(* PLC project pro1003, at09 pro1003 1 *)
(* stored: creationDateTime 2023-04-16T15:18:15, productRelease 0, modificationDateTime 2023-05-21T16:46:51, version 1, language ru-RU *)

(* LED Control *)
PROGRAM prog_led
  VAR_EXTERNAL
    LED_USER : BOOL;
    STATE_REGUL : WORD;
  END_VAR
  VAR
    TONb0 : TONb;
  END_VAR

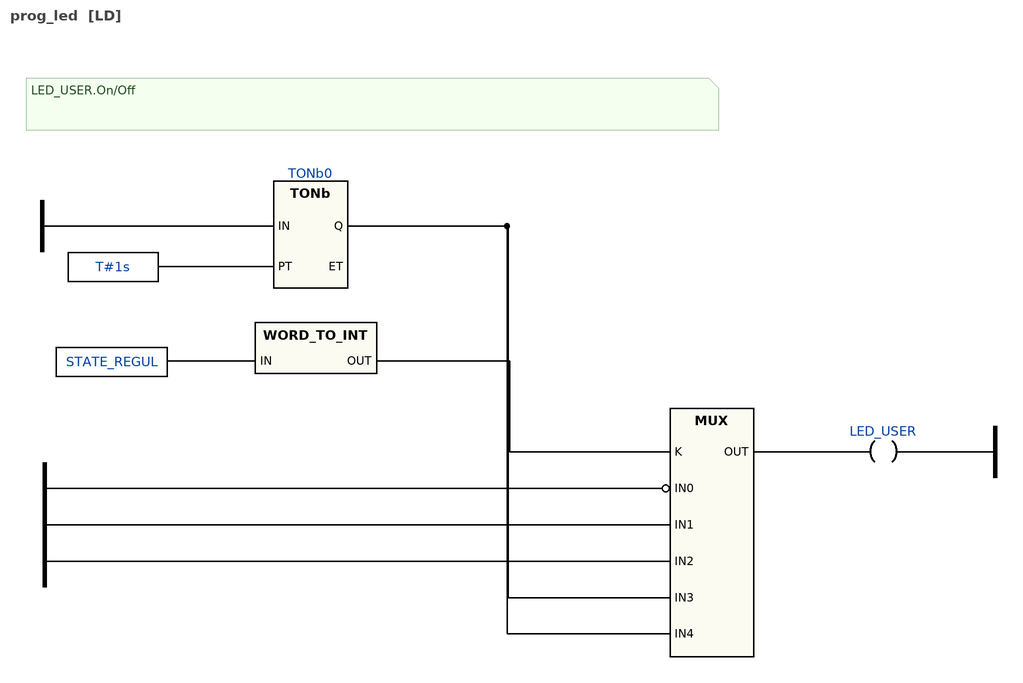
(* LD diagram, written out as Structured Text *)
(* LED_USER.On/Off *)
TONb0(IN := TRUE, PT := T#1s);
LED_USER := MUX(WORD_TO_INT(STATE_REGUL), NOT TRUE, TRUE, TRUE, TONb0.Q, TONb0.Q);
END_PROGRAM

(* Button Control *)
PROGRAM prog_button
  VAR_EXTERNAL CONSTANT
    HS_001_DIn : BYTE;
    HS_002_DIn : BYTE;
  END_VAR
  VAR CONSTANT
    DIMode_Norm : BYTE := 1;  (* DI.Mode (Normal) *)
  END_VAR
  VAR
    DIMode0 : DIMode;
    DIMode1 : DIMode;
  END_VAR

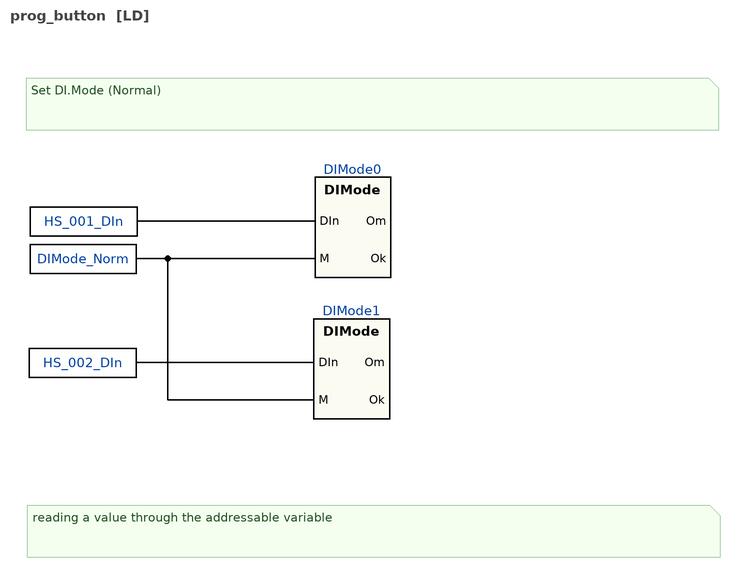
(* LD diagram, written out as Structured Text *)
(* Set DI.Mode (Normal) *)
DIMode0(DIn := HS_001_DIn, M := DIMode_Norm);
DIMode1(DIn := HS_002_DIn, M := DIMode_Norm);
(* reading a value through the addressable variable *)
END_PROGRAM

(* Sensor Control *)
PROGRAM prog_sensor
  VAR_EXTERNAL CONSTANT
    TT_001_AIn : BYTE;
    TT_MCU_AIn2 : BYTE;
  END_VAR
  VAR CONSTANT
    AIMode_Tmp36 : BYTE := 11;  (* AI.Mode (TMP36) *)
    AIMode_TmpMcu : BYTE := 12;  (* AI.Mode (TMP_MCU) *)
  END_VAR
  VAR
    AIMode0 : AIMode;
    AIMode1 : AIMode;
  END_VAR

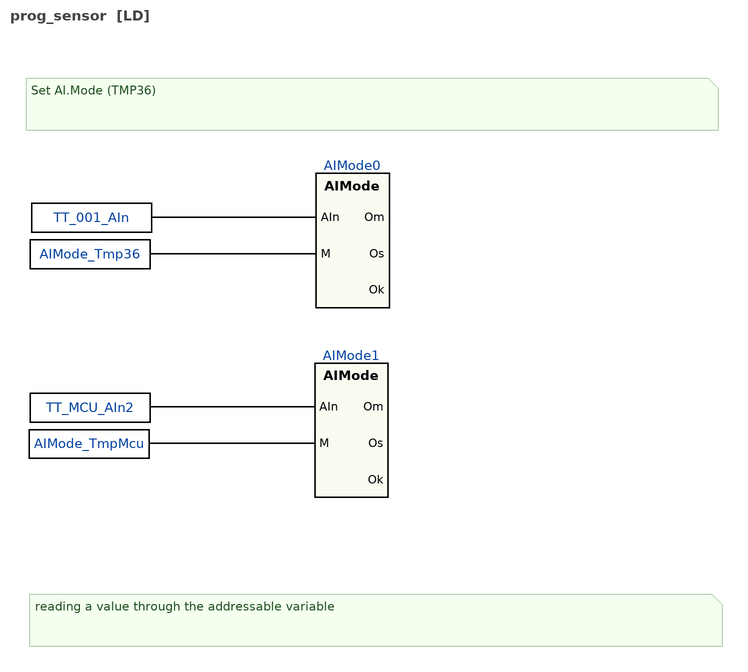
(* LD diagram, written out as Structured Text *)
(* Set AI.Mode (TMP36) *)
AIMode0(AIn := TT_001_AIn, M := AIMode_Tmp36);
AIMode1(AIn := TT_MCU_AIn2, M := AIMode_TmpMcu);
(* reading a value through the addressable variable *)
END_PROGRAM

(* Output Control *)
PROGRAM prog_output
  VAR_EXTERNAL CONSTANT
    H_001_DOn : BYTE;
  END_VAR
  VAR_EXTERNAL
    H_001_V : BOOL;
  END_VAR
  VAR_EXTERNAL CONSTANT
    C_001_DOn : BYTE;
  END_VAR
  VAR_EXTERNAL
    C_001_V : BOOL;
    STATE_REGUL : WORD;
    HEAT : BOOL;
  END_VAR
  VAR CONSTANT
    DOMode_Norm : BYTE := 1;  (* DO.Mode (Normal) *)
  END_VAR
  VAR
    DOMode0 : DOMode;
    DOMode1 : DOMode;
  END_VAR
  VAR  (* added by the conversion: wires and edge detectors of the diagram *)
    _WORD_TO_INT26_OUT : INT;
  END_VAR

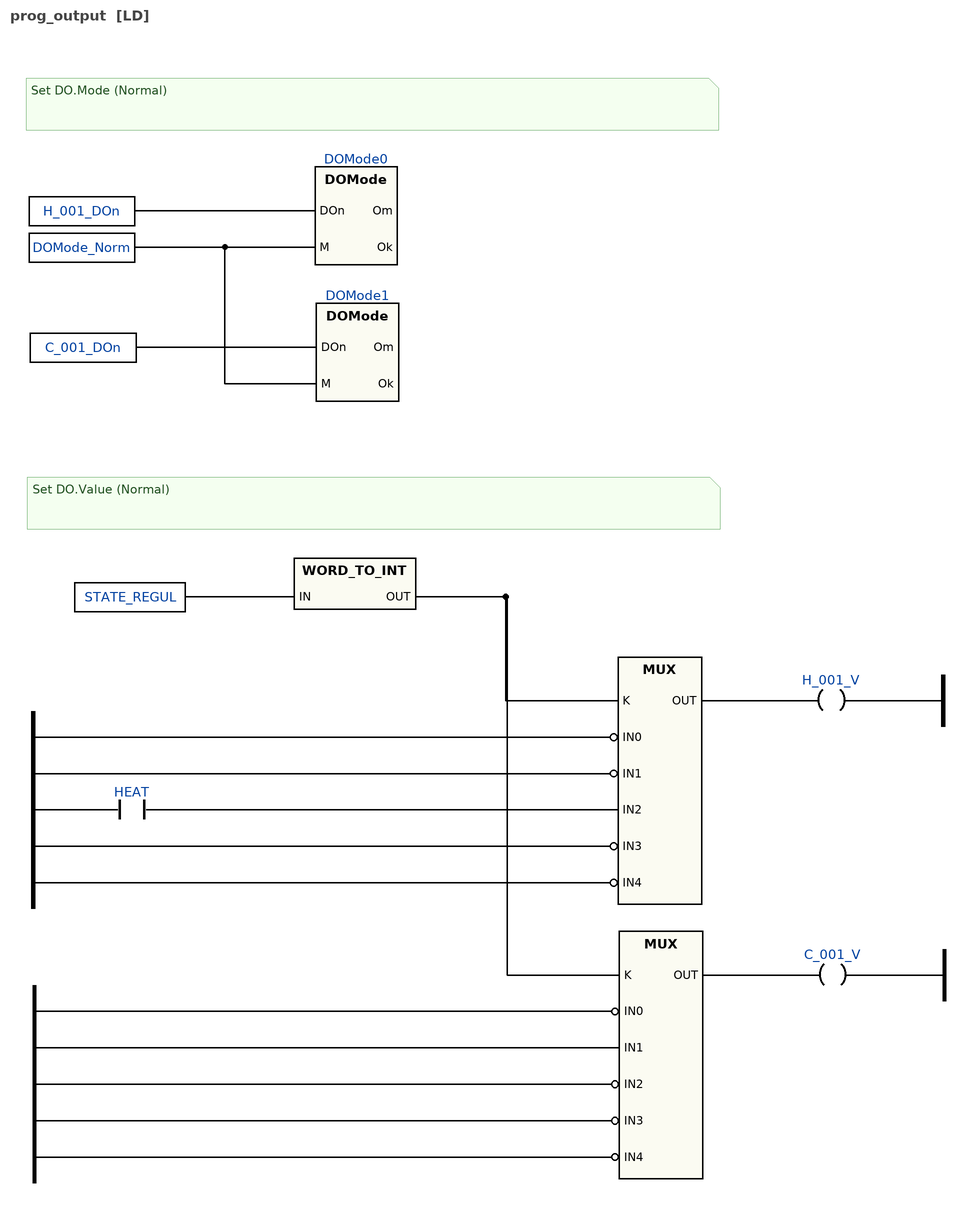
(* LD diagram, written out as Structured Text *)
(* Set DO.Mode (Normal) *)
(* Set DO.Value (Normal) *)
_WORD_TO_INT26_OUT := WORD_TO_INT(STATE_REGUL);
H_001_V := MUX(_WORD_TO_INT26_OUT, NOT TRUE, NOT TRUE, HEAT, NOT TRUE, NOT TRUE);
C_001_V := MUX(_WORD_TO_INT26_OUT, NOT TRUE, TRUE, NOT TRUE, NOT TRUE, NOT TRUE);
DOMode0(DOn := H_001_DOn, M := DOMode_Norm);
DOMode1(DOn := C_001_DOn, M := DOMode_Norm);
END_PROGRAM

(* Regulator *)
PROGRAM prog_regulator
  VAR_EXTERNAL
    TT_001_V : REAL;
    HS_001_V : BOOL;
    HS_002_V : BOOL;
    SET_REGUL_SP : WORD;
    SET_REGUL_D : WORD;
    SET_BLOW_T : WORD;
    STATE_TT : WORD;
  END_VAR
  VAR CONSTANT
    STATE_TT_MUL : REAL := 10.0;
  END_VAR
  VAR_EXTERNAL
    STATE_REGUL : WORD;
  END_VAR
  VAR_EXTERNAL CONSTANT
    STATE_REGUL0 : WORD;
    STATE_REGUL1 : WORD;
    STATE_REGUL2 : WORD;
    STATE_REGUL3 : WORD;
    STATE_REGUL4 : WORD;
  END_VAR
  VAR_EXTERNAL
    START : WORD;
  END_VAR
  VAR CONSTANT
    START0 : WORD := 0;
  END_VAR
  VAR_EXTERNAL
    STARTB : BOOL;
    HEAT : BOOL;
  END_VAR
  VAR
    TONs0 : TONs;
    Reg2p0 : Reg2p;
  END_VAR
  VAR CONSTANT
    HEAT_Delay : TIME := T#1s;
  END_VAR
  VAR  (* added by the conversion: wires and edge detectors of the diagram *)
    R_TRIG1 : R_TRIG;
    F_TRIG2 : F_TRIG;
    _EQ38_OUT : BOOL;
  END_VAR

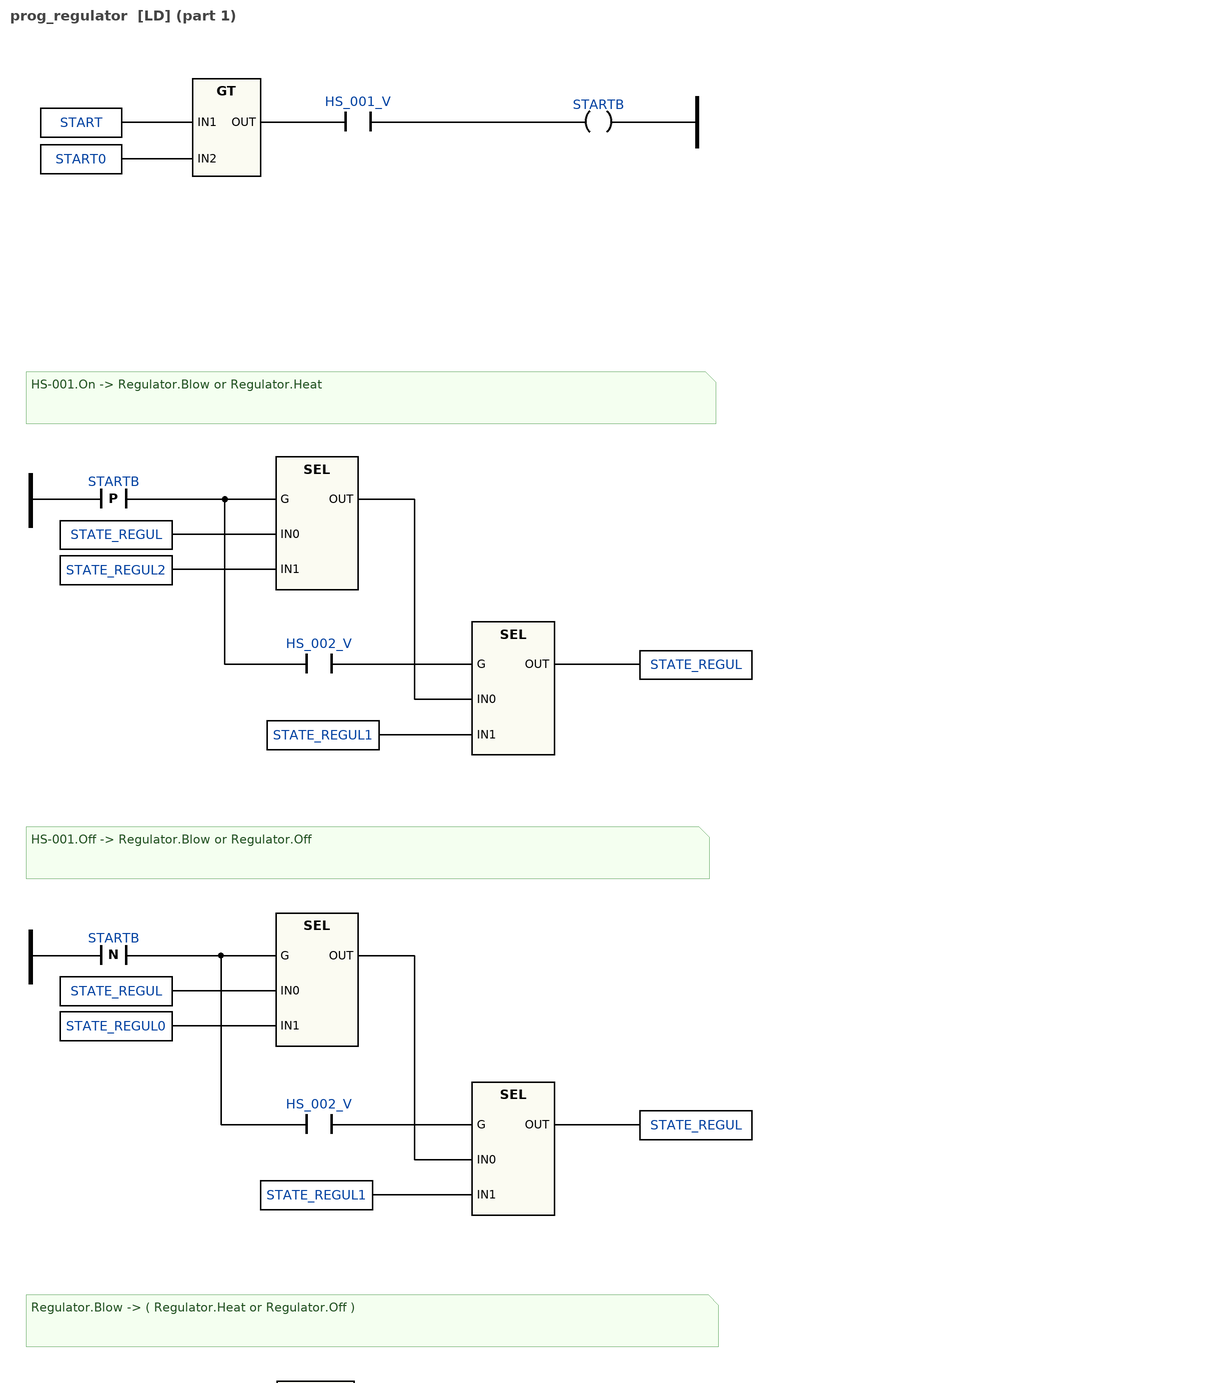
(* LD diagram, written out as Structured Text *)
STARTB := START > START0 AND HS_001_V;
(* HS-001.On -> Regulator.Blow or Regulator.Heat *)
R_TRIG1(CLK := STARTB);
STATE_REGUL := SEL(R_TRIG1.Q AND HS_002_V, SEL(R_TRIG1.Q, STATE_REGUL, STATE_REGUL2), STATE_REGUL1);
(* HS-001.Off -> Regulator.Blow or Regulator.Off *)
F_TRIG2(CLK := STARTB);
STATE_REGUL := SEL(F_TRIG2.Q AND HS_002_V, SEL(F_TRIG2.Q, STATE_REGUL, STATE_REGUL0), STATE_REGUL1);
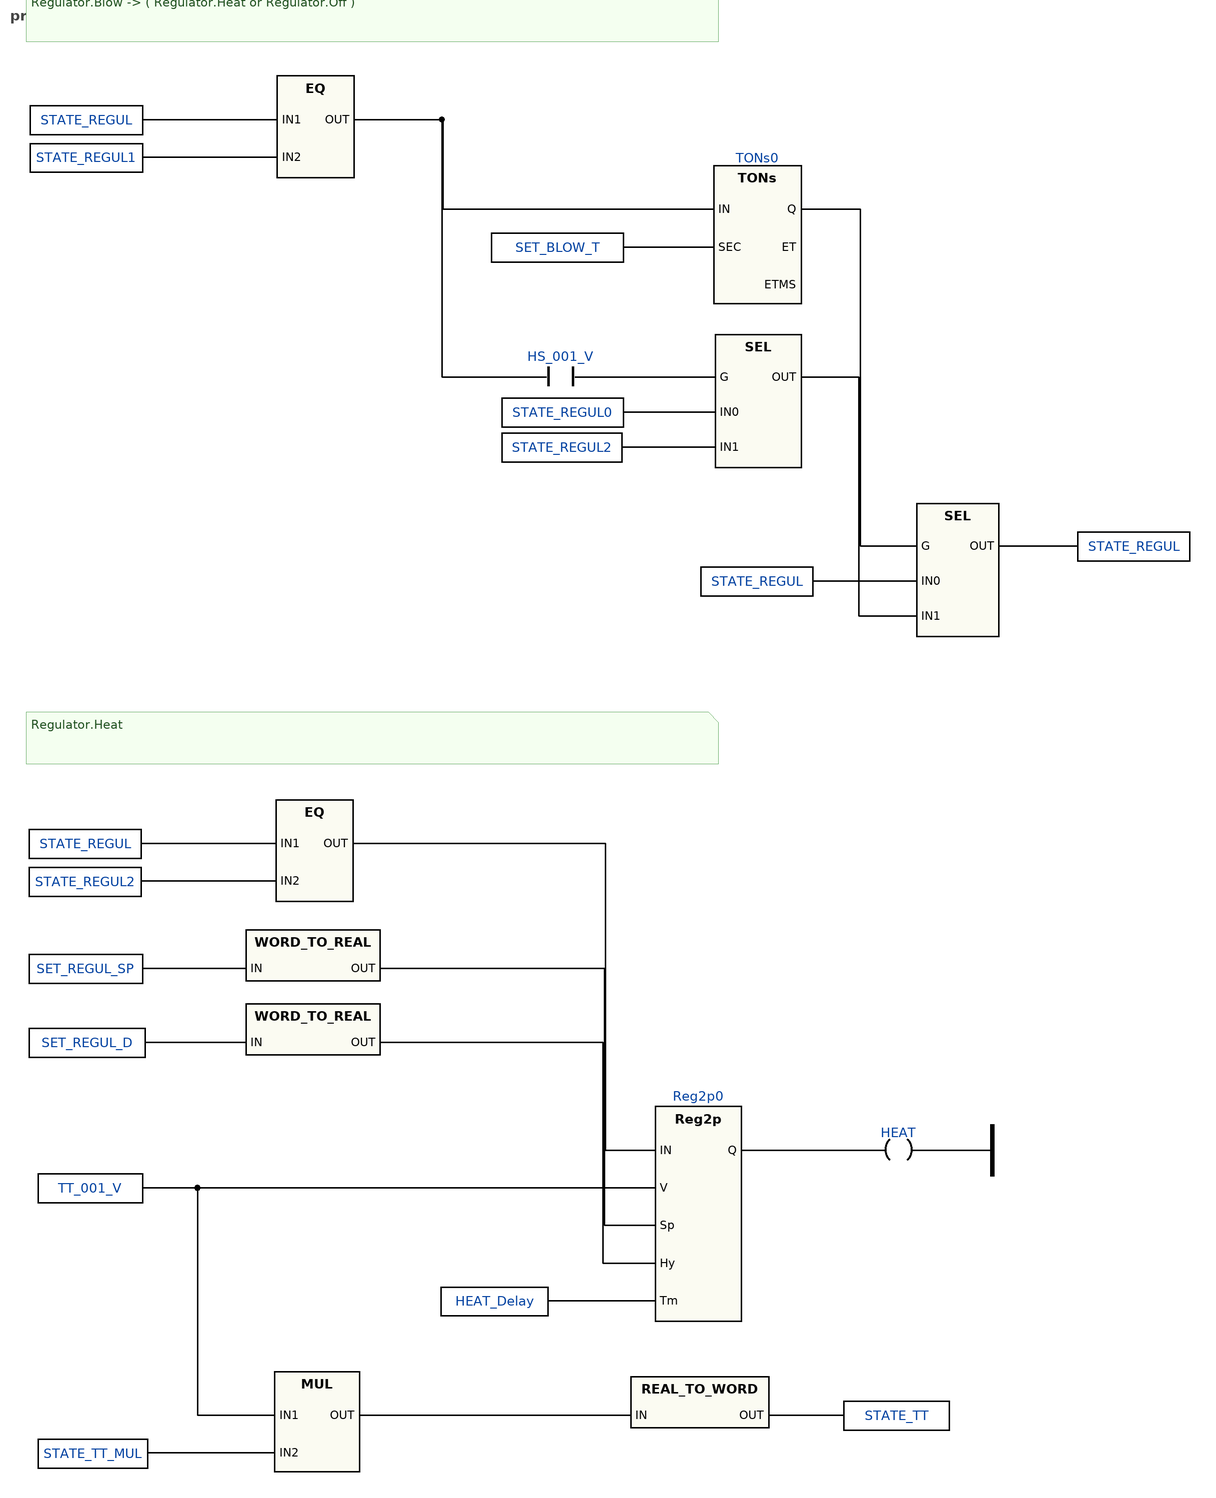
(* Regulator.Blow -> ( Regulator.Heat or Regulator.Off ) *)
_EQ38_OUT := STATE_REGUL = STATE_REGUL1;
TONs0(IN := _EQ38_OUT, SEC := SET_BLOW_T);
STATE_REGUL := SEL(TONs0.Q, STATE_REGUL, SEL(_EQ38_OUT AND HS_001_V, STATE_REGUL0, STATE_REGUL2));
(* Regulator.Heat *)
Reg2p0(IN := STATE_REGUL = STATE_REGUL2, V := TT_001_V, Sp := WORD_TO_REAL(SET_REGUL_SP), Hy := WORD_TO_REAL(SET_REGUL_D), Tm := HEAT_Delay);
HEAT := Reg2p0.Q;
STATE_TT := REAL_TO_WORD(TT_001_V * STATE_TT_MUL);
END_PROGRAM

(* Diagnostic of the Control Loop *)
PROGRAM prog_diagnostic
  VAR_EXTERNAL
    TT_001_V : REAL;
    SET_DIAGN_DHI : WORD;
    SET_DIAGN_THI : WORD;
    SET_DIAGN_DLO : WORD;
    SET_DIAGN_TLO : WORD;
    STATE_REGUL : WORD;
  END_VAR
  VAR_EXTERNAL CONSTANT
    STATE_REGUL3 : WORD;
    STATE_REGUL4 : WORD;
  END_VAR
  VAR_EXTERNAL
    STATE_DIAGN : WORD;
  END_VAR
  VAR_EXTERNAL CONSTANT
    STATE_DIAGN0 : WORD;
    STATE_DIAGN1 : WORD;
    STATE_DIAGN2 : WORD;
  END_VAR
  VAR_EXTERNAL
    HEAT : BOOL;
  END_VAR
  VAR
    LoopCtrl0 : LoopCtrl;
  END_VAR

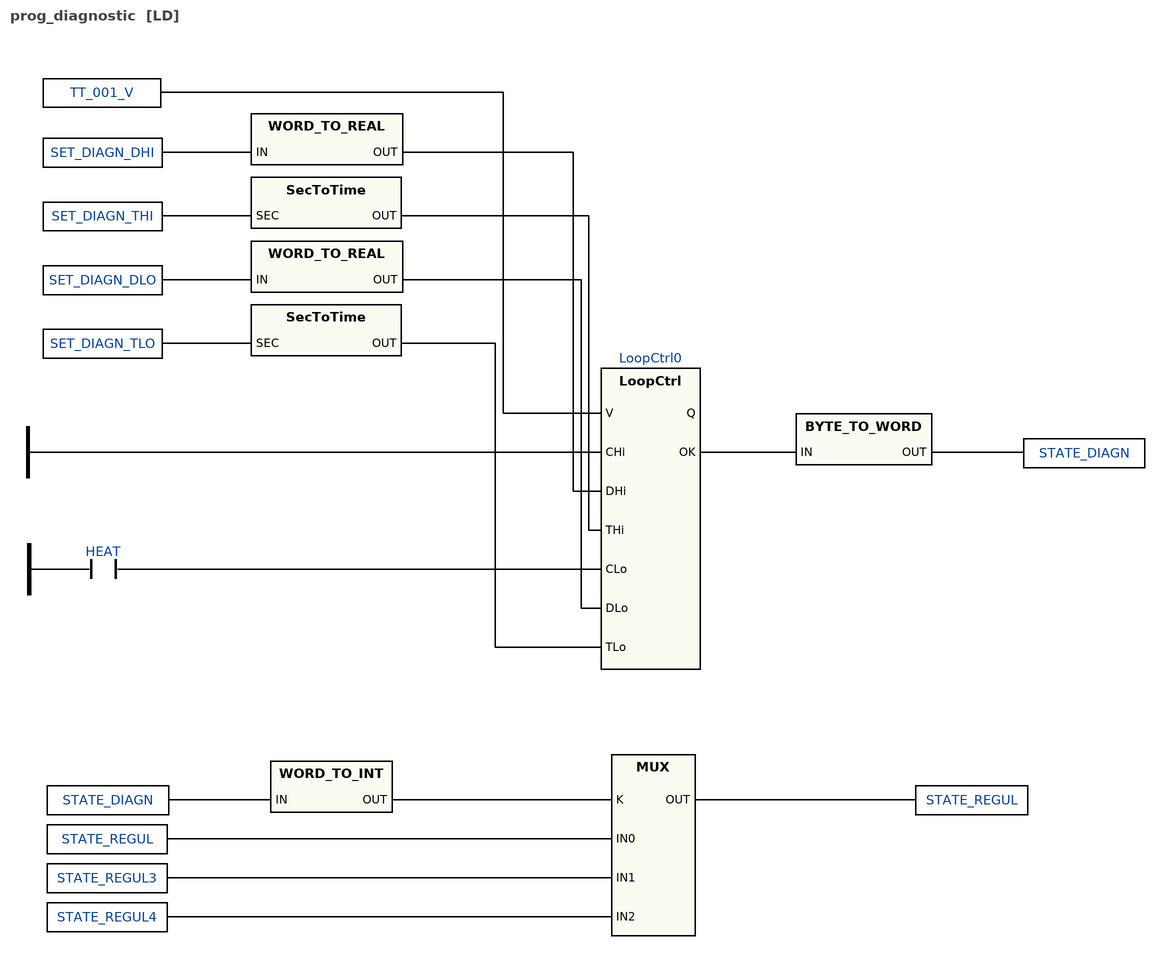
(* LD diagram, written out as Structured Text *)
LoopCtrl0(V := TT_001_V, CHi := TRUE, DHi := WORD_TO_REAL(SET_DIAGN_DHI), THi := SecToTime(SET_DIAGN_THI), CLo := HEAT, DLo := WORD_TO_REAL(SET_DIAGN_DLO), TLo := SecToTime(SET_DIAGN_TLO));
STATE_DIAGN := BYTE_TO_WORD(LoopCtrl0.OK);
STATE_REGUL := MUX(WORD_TO_INT(STATE_DIAGN), STATE_REGUL, STATE_REGUL3, STATE_REGUL4);
END_PROGRAM

(* PLC Pulse *)
PROGRAM prog_pulse
  VAR_EXTERNAL
    TT_MCU_V : REAL;
    PLC : WORD;
    PLC_TT : WORD;
  END_VAR
  VAR CONSTANT
    PLC_TT_MUL : REAL := 10.0;
  END_VAR

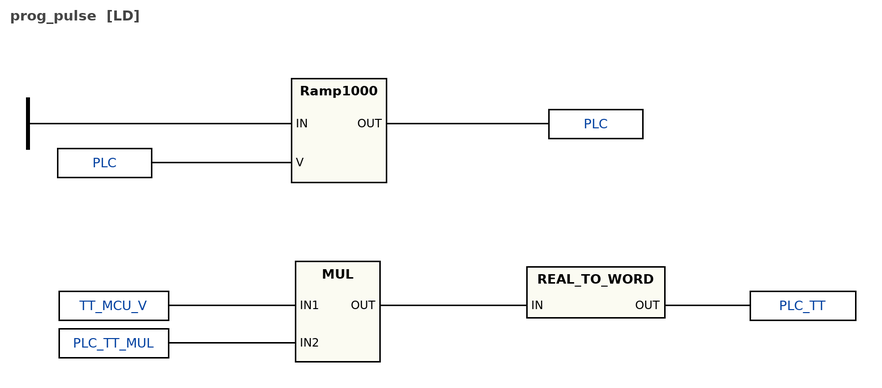
(* LD diagram, written out as Structured Text *)
PLC := Ramp1000(TRUE, PLC);
PLC_TT := REAL_TO_WORD(TT_MCU_V * PLC_TT_MUL);
END_PROGRAM

(* Pack bit-values into STATE-word *)
PROGRAM prog_states
  VAR_EXTERNAL
    HS_001_V : BOOL;
    HS_002_V : BOOL;
    H_001_V : BOOL;
    C_001_V : BOOL;
    LED_USER : BOOL;
    STATE_REGUL : WORD;
  END_VAR
  VAR_EXTERNAL CONSTANT
    STATE_REGUL3 : WORD;
  END_VAR
  VAR_EXTERNAL
    STATES : WORD;
    INIT : BOOL;
  END_VAR

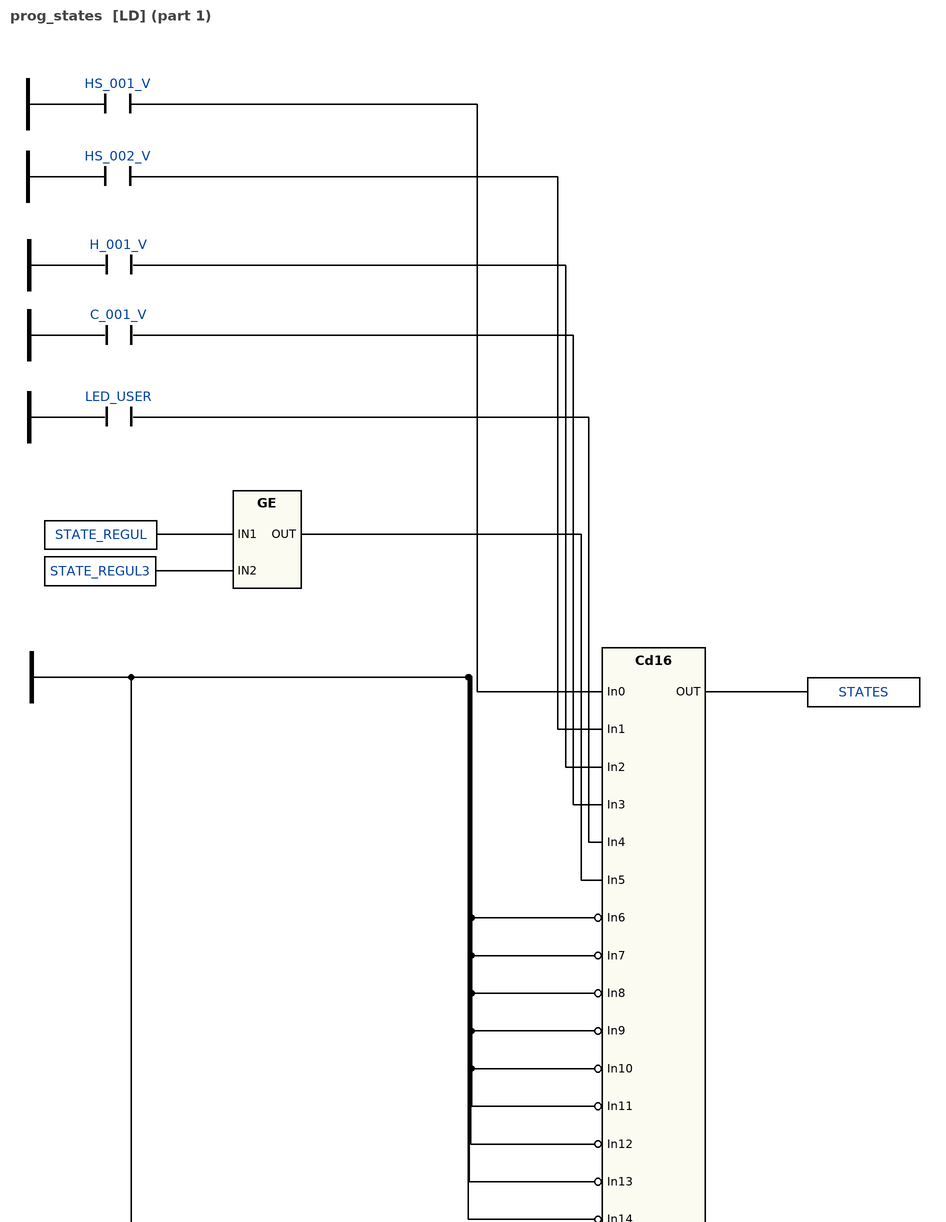
(* LD diagram, written out as Structured Text *)
STATES := Cd16(HS_001_V, HS_002_V, H_001_V, C_001_V, LED_USER, STATE_REGUL >= STATE_REGUL3, NOT TRUE, NOT TRUE, NOT TRUE, NOT TRUE, NOT TRUE, NOT TRUE, NOT TRUE, NOT TRUE, NOT TRUE, INIT);
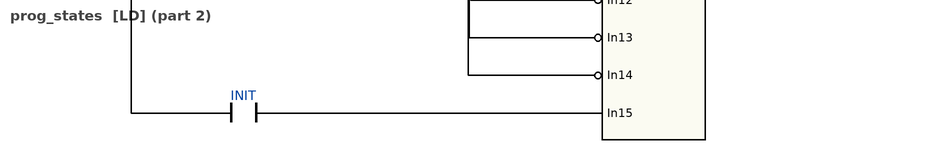
END_PROGRAM

PROGRAM prog_init
  VAR_EXTERNAL
    SET_REGUL_SP : WORD;
  END_VAR
  VAR CONSTANT
    SET_REGUL_SP_DEF : WORD := 40;
  END_VAR
  VAR_EXTERNAL
    SET_REGUL_D : WORD;
  END_VAR
  VAR CONSTANT
    SET_REGUL_D_DEF : WORD := 2;
  END_VAR
  VAR_EXTERNAL
    SET_DIAGN_DHI : WORD;
  END_VAR
  VAR CONSTANT
    SET_DIAGN_DHI_DEF : WORD := 50;
  END_VAR
  VAR_EXTERNAL
    SET_DIAGN_THI : WORD;
  END_VAR
  VAR CONSTANT
    SET_DIAGN_THI_DEF : WORD := 60;  (* sec *)
  END_VAR
  VAR_EXTERNAL
    SET_DIAGN_DLO : WORD;
  END_VAR
  VAR CONSTANT
    SET_DIAGN_DLO_DEF : WORD := 35;
  END_VAR
  VAR_EXTERNAL
    SET_DIAGN_TLO : WORD;
  END_VAR
  VAR CONSTANT
    SET_DIAGN_TLO_DEF : WORD := 300;  (* sec *)
  END_VAR
  VAR_EXTERNAL
    SET_BLOW_T : WORD;
  END_VAR
  VAR CONSTANT
    SET_BLOW_T_DEF : WORD := 60;  (* sec *)
  END_VAR
  VAR_EXTERNAL
    INIT : BOOL;
  END_VAR

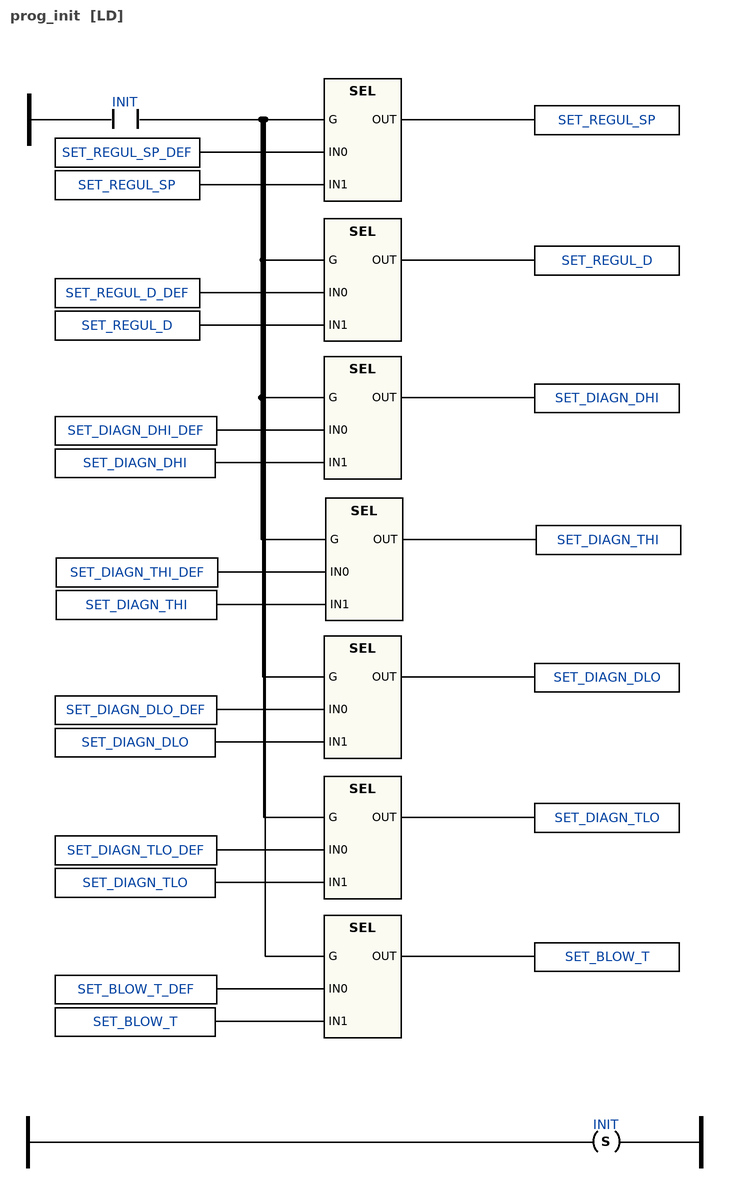
(* LD diagram, written out as Structured Text *)
SET_REGUL_SP := SEL(INIT, SET_REGUL_SP_DEF, SET_REGUL_SP);
SET_REGUL_D := SEL(INIT, SET_REGUL_D_DEF, SET_REGUL_D);
SET_DIAGN_DHI := SEL(INIT, SET_DIAGN_DHI_DEF, SET_DIAGN_DHI);
SET_DIAGN_THI := SEL(INIT, SET_DIAGN_THI_DEF, SET_DIAGN_THI);
SET_DIAGN_DLO := SEL(INIT, SET_DIAGN_DLO_DEF, SET_DIAGN_DLO);
SET_DIAGN_TLO := SEL(INIT, SET_DIAGN_TLO_DEF, SET_DIAGN_TLO);
SET_BLOW_T := SEL(INIT, SET_BLOW_T_DEF, SET_BLOW_T);
IF TRUE THEN INIT := TRUE; END_IF;
END_PROGRAM

CONFIGURATION config
  VAR_GLOBAL CONSTANT
    HS_001_DIn : BYTE := 0;  (* DI.Channel *)
  END_VAR
  VAR_GLOBAL
    HS_001_V AT %IX1.0.1.1 : BOOL := FALSE;  (* DI.Value (Normal) *)
  END_VAR
  VAR_GLOBAL CONSTANT
    HS_002_DIn : BYTE := 1;  (* DI.Channel *)
  END_VAR
  VAR_GLOBAL
    HS_002_V AT %IX1.1.1.1 : BOOL := FALSE;  (* DI.Value (Normal) *)
  END_VAR
  VAR_GLOBAL CONSTANT
    TT_001_AIn : BYTE := 0;  (* AI.Channel *)
  END_VAR
  VAR_GLOBAL
    TT_001_V AT %ID3.0.1 : REAL := 0.0;  (* AI.Value (grad. C) *)
  END_VAR
  VAR_GLOBAL CONSTANT
    TT_MCU_AIn2 : BYTE := 2;  (* AI.Channel *)
  END_VAR
  VAR_GLOBAL
    TT_MCU_V AT %ID3.2.1 : REAL := 0.0;  (* AI.Value (grad. C) *)
  END_VAR
  VAR_GLOBAL CONSTANT
    H_001_DOn : BYTE := 0;  (* DO.Channel *)
  END_VAR
  VAR_GLOBAL
    H_001_V AT %QX2.0.1.1 : BOOL := FALSE;  (* DO.Value (Normal) *)
  END_VAR
  VAR_GLOBAL CONSTANT
    C_001_DOn : BYTE := 1;  (* DO.Channel *)
  END_VAR
  VAR_GLOBAL
    C_001_V AT %QX2.1.1.1 : BOOL := FALSE;  (* DO.Value (Normal) *)
    LED_USER AT %MX7.3.0 : BOOL := FALSE;  (* LED_USER.On/Off *)
    SET_REGUL_SP AT %MW8.2.1 : WORD := 0;  (* Settings.Regulator.Setpoint (grad. C) *)
    SET_REGUL_D AT %MW8.2.2 : WORD := 0;  (* Settings.Regulator.Hysteresis (grad. C) *)
    SET_DIAGN_DHI AT %MW8.2.3 : WORD := 0;  (* Settings.LoopControl.Hysteresis (grad. C) *)
    SET_DIAGN_THI AT %MW8.2.4 : WORD := 0;  (* Settings.LoopControl.DelayTime (sec) *)
    SET_DIAGN_DLO AT %MW8.2.5 : WORD := 0;  (* Settings.LoopControl.DelayTime (sec) *)
    SET_DIAGN_TLO AT %MW8.2.6 : WORD := 0;  (* Settings.LoopControl.DelayTime (sec) *)
    SET_BLOW_T AT %MW8.2.7 : WORD := 0;  (* Settings.Blow.Time (sec) *)
    STATES AT %MW8.2.8 : WORD := 0;  (* Output.States (bitfield) *)
    STATE_TT AT %MW8.2.9 : WORD := 0;  (* Output.Temp (grad. C) *)
    STATE_REGUL AT %MW8.2.10 : WORD := 0;  (* Regulator.StateCode (0 - Off, 1 - Blow, 2 - Heat, 3 - Low Zone alarm, 4 - High Zone alarm) *)
  END_VAR
  VAR_GLOBAL CONSTANT
    STATE_REGUL0 : WORD := 0;  (* Regulator.Off *)
    STATE_REGUL1 : WORD := 1;  (* Regulator.Blow *)
    STATE_REGUL2 : WORD := 2;  (* Regulator.Work *)
    STATE_REGUL3 : WORD := 3;  (* Regulator.LowZoneAlarm *)
    STATE_REGUL4 : WORD := 4;  (* Regulator.HighZoneAlarm *)
  END_VAR
  VAR_GLOBAL
    STATE_DIAGN AT %MW8.2.11 : WORD := 0;  (* Diagnostic.StateCode (0 - Normal, 1 - Low Zone alarm, 2 - High Zone alarm) *)
  END_VAR
  VAR_GLOBAL CONSTANT
    STATE_DIAGN0 : WORD := 0;  (* Diagnostic.Normal *)
    STATE_DIAGN1 : WORD := 1;  (* Diagnostic.LowZone *)
    STATE_DIAGN2 : WORD := 2;  (* Diagnostic.HighZone *)
  END_VAR
  VAR_GLOBAL
    PLC AT %MW8.2.12 : WORD := 0;  (* PLC.Pulse *)
    PLC_TT AT %MW8.2.13 : WORD := 0;  (* PLC.MCU_TEMP *)
    START AT %MW8.2.14 : WORD := 0;  (* Remote command: 0 - Stop, >0 - Start *)
    STARTB : BOOL := FALSE;  (* Remote command: FALSE - Stop, TRUE - Start *)
    HEAT : BOOL := FALSE;  (* Requlator.Heat (output) *)
    INIT : BOOL := FALSE;  (* First initialization flag (0 - not inited, 1 - inited) *)
  END_VAR
  RESOURCE resource1 ON PLC
    TASK task0(INTERVAL := T#300ms, PRIORITY := 0);
    PROGRAM instance0 WITH task0 : prog_init;
    PROGRAM instance1 WITH task0 : prog_button;
    PROGRAM instance2 WITH task0 : prog_sensor;
    PROGRAM instance3 WITH task0 : prog_regulator;
    PROGRAM instance5 WITH task0 : prog_pulse;
    PROGRAM instance6 WITH task0 : prog_states;
    PROGRAM instance7 WITH task0 : prog_output;
    PROGRAM instance8 WITH task0 : prog_led;
  END_RESOURCE
END_CONFIGURATION
